# B&R Automation Studio project SFL4_230526
Automation Studio 4.9.2.46; technology packages: mapp 5.12.0

## Configuration Config1

CPU 4PPC70.0702-20B, AutomationRuntime C4.90, Build 4.1.2, Vc V4.72.2

### Task classes (Cpu.sw)
```
Cyclic#4:
  Program <- Program.prg
Libraries: MpDatabase, MpBase, AsHttp, runtime
```

### Hardware
```
4PPC70_0702_20B : 4PPC70.0702-20B v1.5.2.0
  Connector IF2:
    ActivateDevice = 1
    Mode = Manual
    InternetAddress = 10.16.7.86
    SubnetMask = 255.255.0.0
    ActivateSnmp = 2
  ConfigurationID = SFL4_230526_Config1
  KeyMappingFile = VC\4PPC70_0702_20B.dis
```

### Config.mpdatabasecore - 4PPC70_0702_20B/mappServices/Config.mpdatabasecore
```
Element gDatabaseCore (Type=mpdatabasecore)
  mapp.Database.Core:
    Name = manitou
    UserName = Manitou
    Password = Ganz_Wien79
    IPAddress = 10.16.7.86
    PortNumber = 3306
```

## Logical view

Binary libraries used (declarations not repeated): operator, runtime, astime, AsIecCon, MpDatabase 5.12.0, MpBase, AsHttp

### Program Logical/Program

#### Variables.var
```iecst
VAR
	MpDatabaseCore_0 : MpDatabaseCore;
	MpDatabaseQuery_0 : MpDatabaseQuery;
END_VAR
```

#### Cyclic.ld
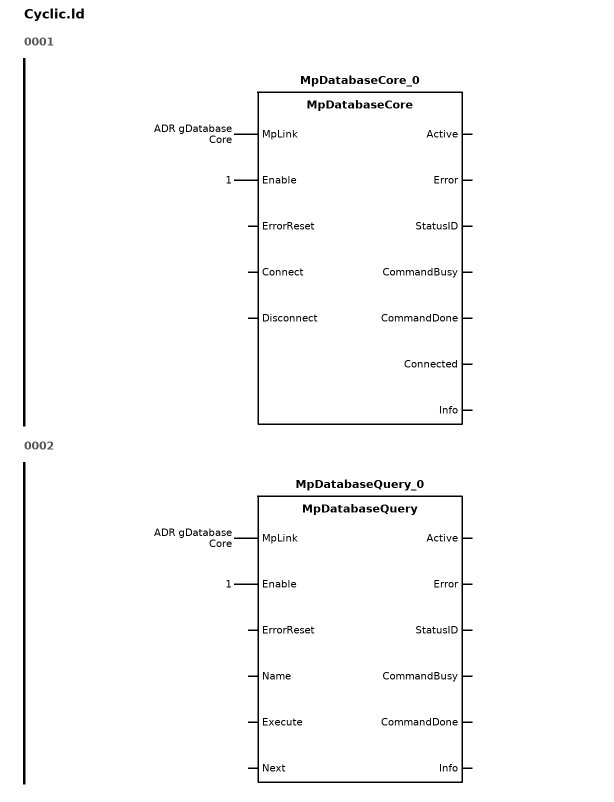
Ladder, written as Structured Text:
```iecst
PROGRAM _CYCLIC
(* Network 1 *)
MpDatabaseCore_0(MpLink := ADR(gDatabaseCore), Enable := 1);

(* Network 2 *)
MpDatabaseQuery_0(MpLink := ADR(gDatabaseCore), Enable := 1);
END_PROGRAM
```

#### Exit.ld
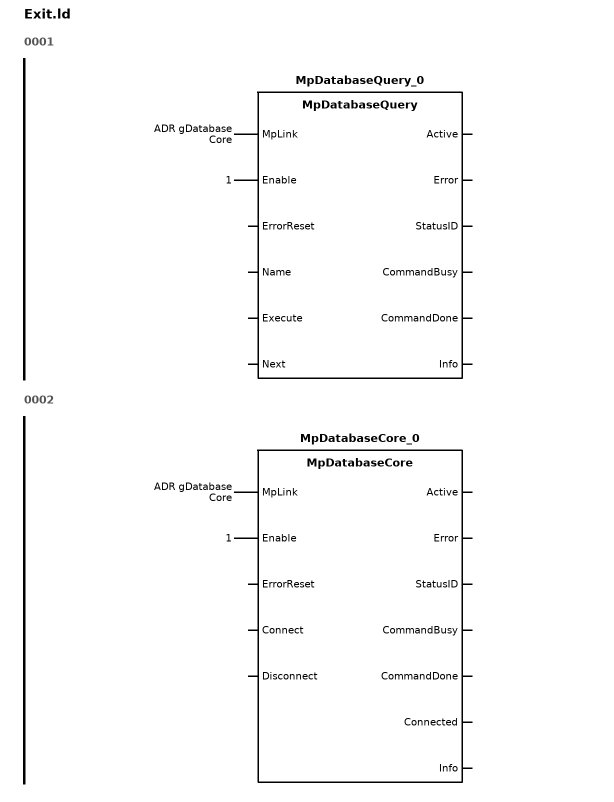
Ladder, written as Structured Text:
```iecst
PROGRAM _EXIT
(* Network 1 *)
MpDatabaseQuery_0(MpLink := ADR(gDatabaseCore), Enable := 1);

(* Network 2 *)
MpDatabaseCore_0(MpLink := ADR(gDatabaseCore), Enable := 1);
END_PROGRAM
```

#### Init.ld
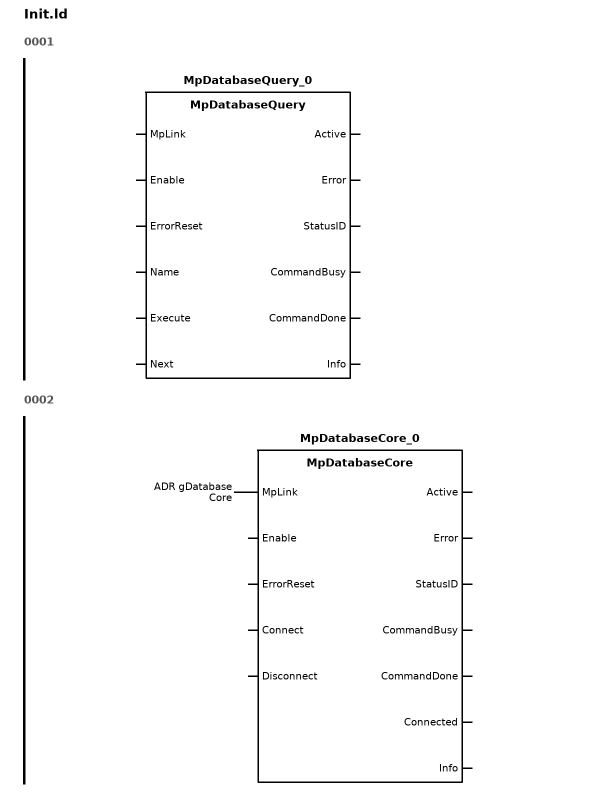
Ladder, written as Structured Text:
```iecst
PROGRAM _INIT
(* Network 1 *)
MpDatabaseQuery_0();

(* Network 2 *)
MpDatabaseCore_0(MpLink := ADR(gDatabaseCore));
END_PROGRAM
```
